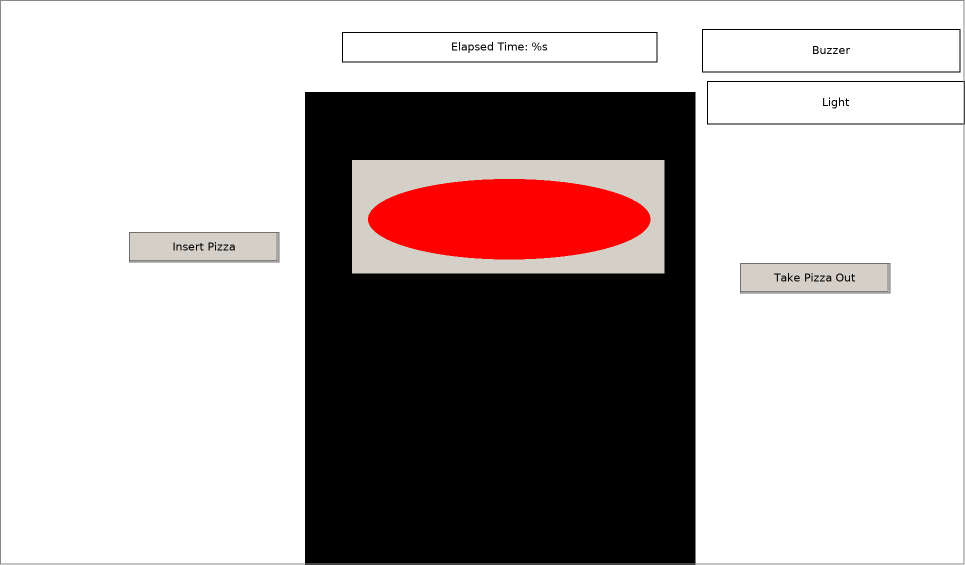
VISUALIZATION Visualization  // 965x565
    Button (129,232 150x30), "Insert Pizza"
        OnMouseClick: execute { MAIN.bPizzaInOven := TRUE; }
    Button (740,263 150x30), "Take Pizza Out"
        OnMouseClick: execute { MAIN.bPizzaInOver := False; }
    Rectangle (305,92 390x473)
    Rectangle (342,32 315x30), "Elapsed Time: %s", text variable: MAIN.fbPizzaTimer.ET
    RoundedRectangle (352,160 312x113)
    Ellipse (367,178 284x82), invisible if: NOT MAIN.bPizzaInOven
    RoundedRectangle (702,29 258x43), "Buzzer", colour toggle: MAIN.bBuzzer
    RoundedRectangle (707,81 258x43), "Light", colour toggle: MAIN.bPizzaInOven
END_VISUALIZATION

(* stored: Version 1.1.0.1, ProductVersion 3.1.4024.16
   Visu Visualization: Id {0d3eb007-1c4c-411c-b1ba-4f2c9d64b5e9} *)
